Yaskawa INFORM job: TESTJOB2.JBI

/JOB
//NAME TESTJOB2
//POS
///NPOS 0,0,0,2,0,0
///TOOL 0
///POSTYPE PULSE
///PULSE
P00000=0,0,0,0,0,0
///USER 1
///POSTYPE USER
///RECTAN
///RCONF 0,0,0,0,0,0,0,0,0,0,0,0,0,0,0,0,0,0,0,0,0,0,0,0
P00003=300.000,0.000,0.000,0.0000,0.0000,0.0000
//INST
///DATE 2010/10/22 11:18
///ATTR SC,RW
///GROUP1 RB1
NOP
MOVL P000 V=33.3
MOVL P003 V=33.3
END
